TYPE ST_VG :
STRUCT
	/// A general gauge structure is used to make the rest of the interlocking simpler. There are some parameters for cold cathodes that are not used by pirani.
	///These features aren't disabled, they just aren't used, think child/parent classes. 
	/// Readbacks 
	rPRESS: REAL; //This is the human-readable pressure
	iPRESS_R: INT; //input pressure in machine form
	xAT_VAC: BOOL; //Pressure At Vacuum
	xPRESS_OK: BOOL; // Pressure Reading is trustworthy
	wState	:	WORD; //current gauge state, to be used as replacement for press OK bit in the future.
	(* 00 controller not on
		01 normal, aka pressure OK
		02 LO, pressure too low
		03 HI, pressure too high
		04 Gauge disconnected, HV off, no sensor detected, controller powering up
		05 cold cathode warming up
		*)
	eState	:	E_PressureState;
	
	/// Controls 
	xHV_DIS: BOOL;// Enable High Voltage when True
	xHV_SW: BOOL;// High Voltage Switch
	wHV_RO: WORD;// Relay Output Location
	
	xBAKEOUT: BOOL; /// Bakeout bit 
	
	eTYPE: Gauge_Type := PG907; //enum for gauge type
	iTYPE : INT := 0;
	wPG: WORD;  /// Index location of the associated Pirani Guage
	
	xTurnOnTime: BOOL;/// Turn on Timers for cold cathode warmup 
	
	rVAC_SP: REAL := 0.5; // At vacuum setpoint for all gauges
	rPRO_SP: REAL := 0.01; // Protection setpoint for ion gauges at which the gauge turns off, not used for pirani
	rHYS_PR: REAL; // Protection setpoint hysteresis 
	rFULL_SCALE: REAL := 1000; // Full scale pressure in Torr for baratron pressure conversion 
END_STRUCT
END_TYPE

(* stored: Version 1.1.0.1, ProductVersion 3.1.4018.5
   DUT ST_VG: Id {8ebcc563-a05a-4cb9-b161-a02f8eac0f57} *)
